// SIMATIC S7-200 project (STEP 7-Micro/WIN), CPU 224 UN REL 02.01

ORGANIZATION_BLOCK 主程序:OB1
TITLE=程序注释
BEGIN
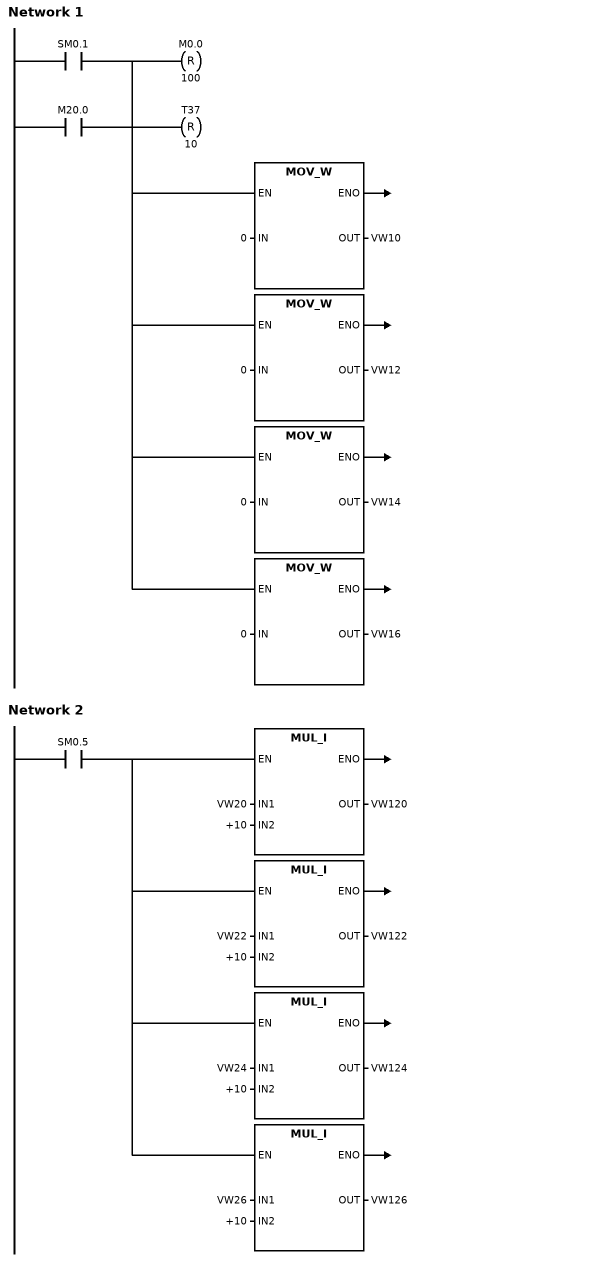
Network 1
LD     SM0.1
O      M20.0
R      M0.0, 100
R      T37, 10
MOVW   0, VW10
MOVW   0, VW12
MOVW   0, VW14
MOVW   0, VW16
Network 2
LD     SM0.5
MOVW   VW20, VW120
*I     +10, VW120
MOVW   VW22, VW122
*I     +10, VW122
MOVW   VW24, VW124
*I     +10, VW124
MOVW   VW26, VW126
*I     +10, VW126
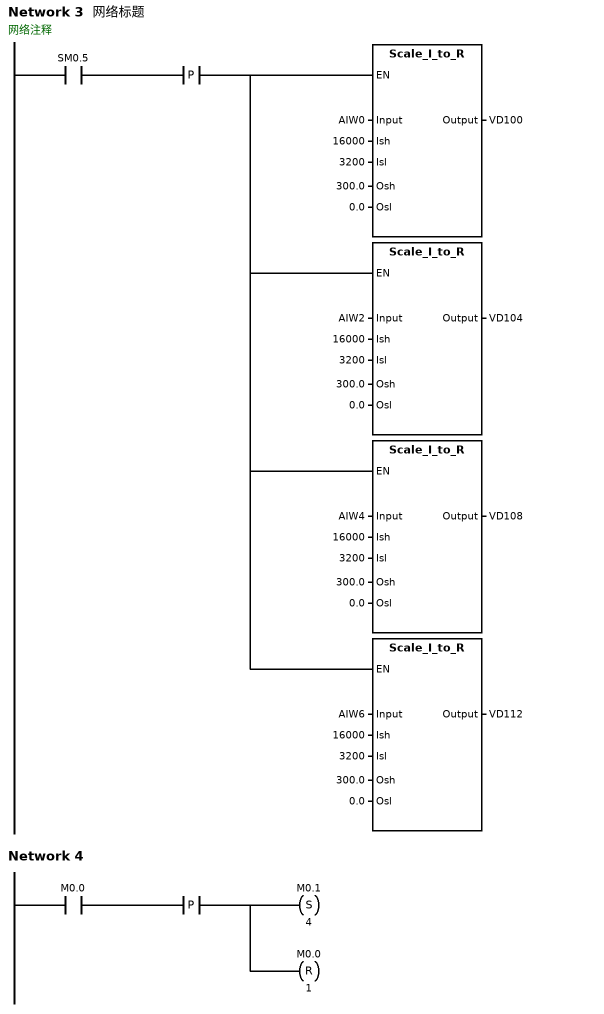
Network 3 // 网络标题
// 网络注释
LD     SM0.5
EU
CALL   Scale_I_to_R:SBR1, AIW0, 16000, 3200, 300.0, 0.0, VD100
CALL   Scale_I_to_R:SBR1, AIW2, 16000, 3200, 300.0, 0.0, VD104
CALL   Scale_I_to_R:SBR1, AIW4, 16000, 3200, 300.0, 0.0, VD108
CALL   Scale_I_to_R:SBR1, AIW6, 16000, 3200, 300.0, 0.0, VD112
Network 4
LD     M0.0
EU
S      M0.1, 4
R      M0.0, 1
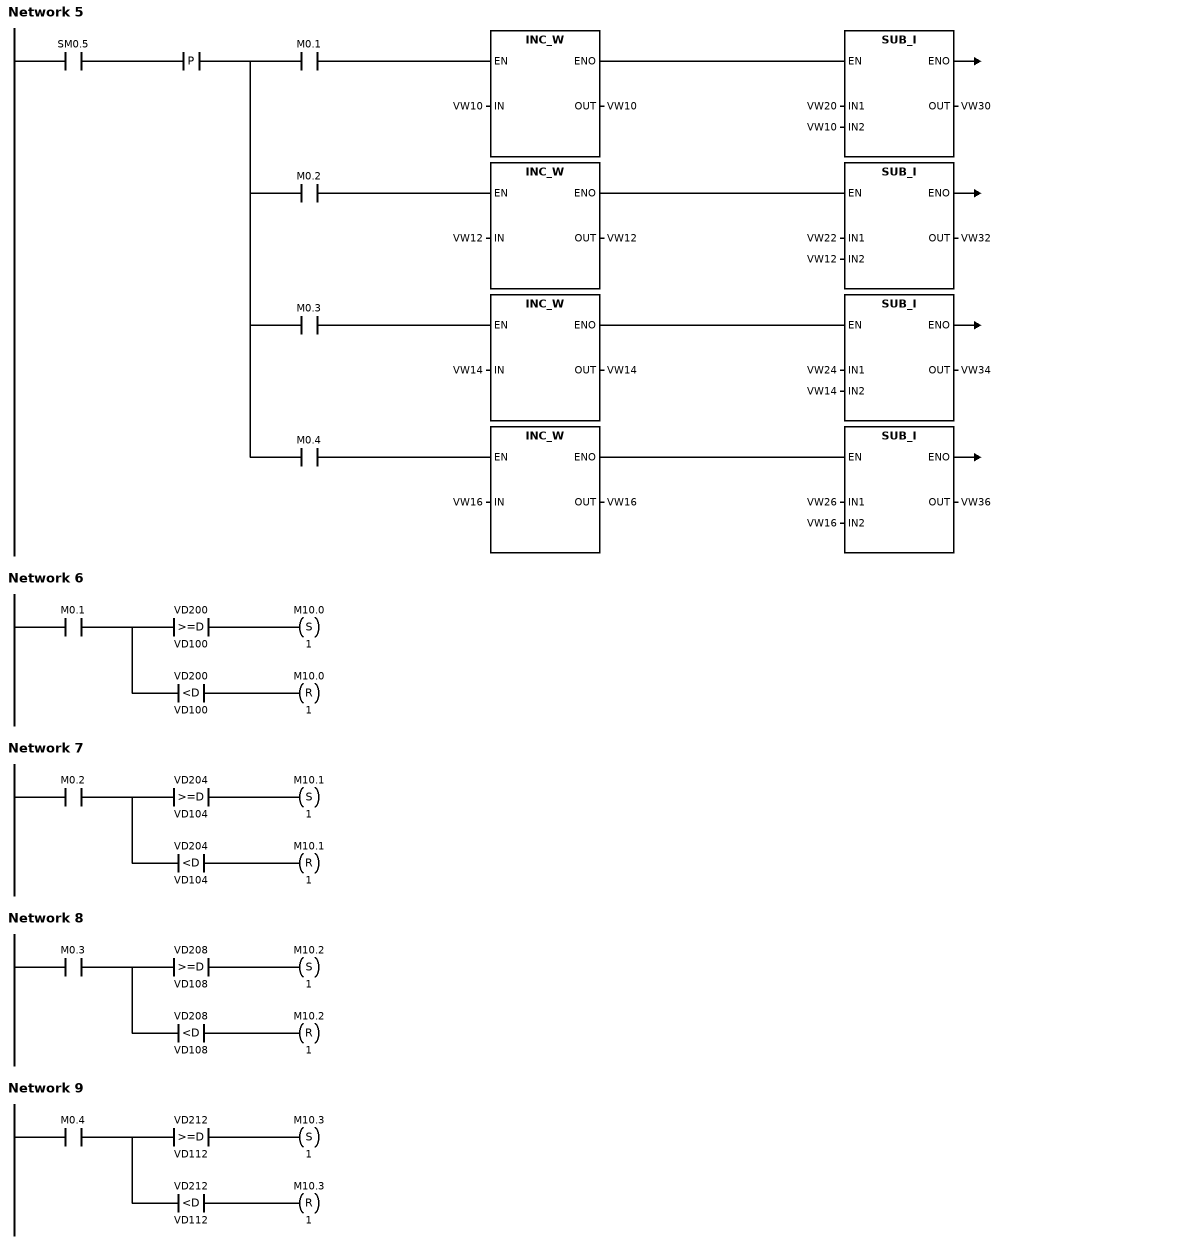
Network 5
LD     SM0.5
EU
LPS
A      M0.1
INCW   VW10
AENO
MOVW   VW20, VW30
-I     VW10, VW30
LRD
A      M0.2
INCW   VW12
AENO
MOVW   VW22, VW32
-I     VW12, VW32
LRD
A      M0.3
INCW   VW14
AENO
MOVW   VW24, VW34
-I     VW14, VW34
LPP
A      M0.4
INCW   VW16
AENO
MOVW   VW26, VW36
-I     VW16, VW36
Network 6
LD     M0.1
LPS
AD>=   VD200, VD100
S      M10.0, 1
LPP
AD<    VD200, VD100
R      M10.0, 1
Network 7
LD     M0.2
LPS
AD>=   VD204, VD104
S      M10.1, 1
LPP
AD<    VD204, VD104
R      M10.1, 1
Network 8
LD     M0.3
LPS
AD>=   VD208, VD108
S      M10.2, 1
LPP
AD<    VD208, VD108
R      M10.2, 1
Network 9
LD     M0.4
LPS
AD>=   VD212, VD112
S      M10.3, 1
LPP
AD<    VD212, VD112
R      M10.3, 1
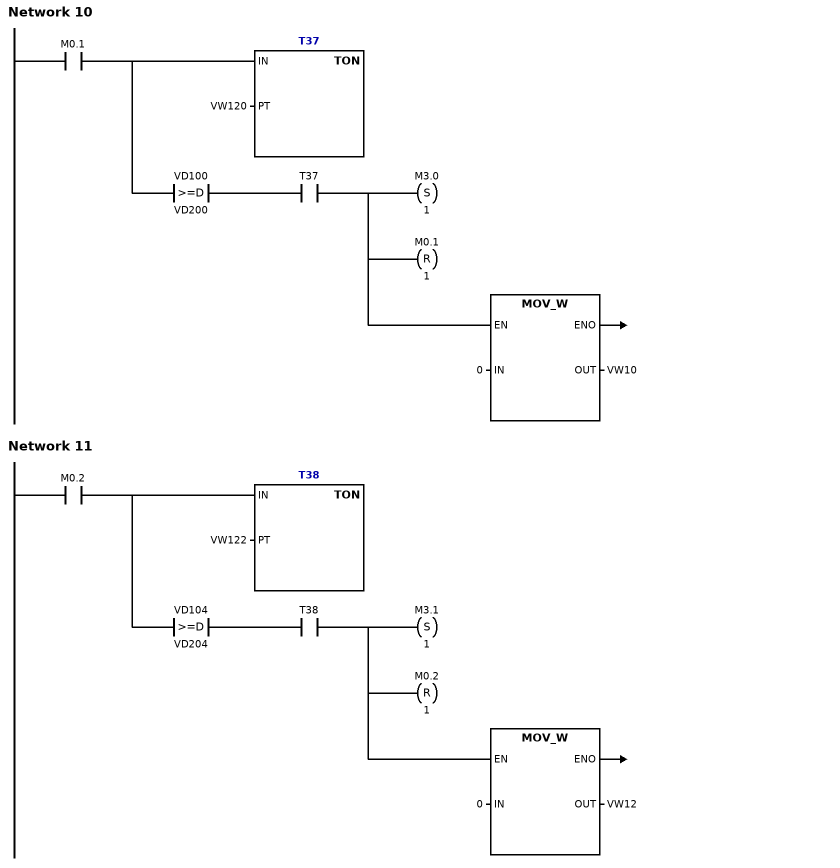
Network 10
LD     M0.1
TON    T37, VW120
AD>=   VD100, VD200
A      T37
S      M3.0, 1
R      M0.1, 1
MOVW   0, VW10
Network 11
LD     M0.2
TON    T38, VW122
AD>=   VD104, VD204
A      T38
S      M3.1, 1
R      M0.2, 1
MOVW   0, VW12
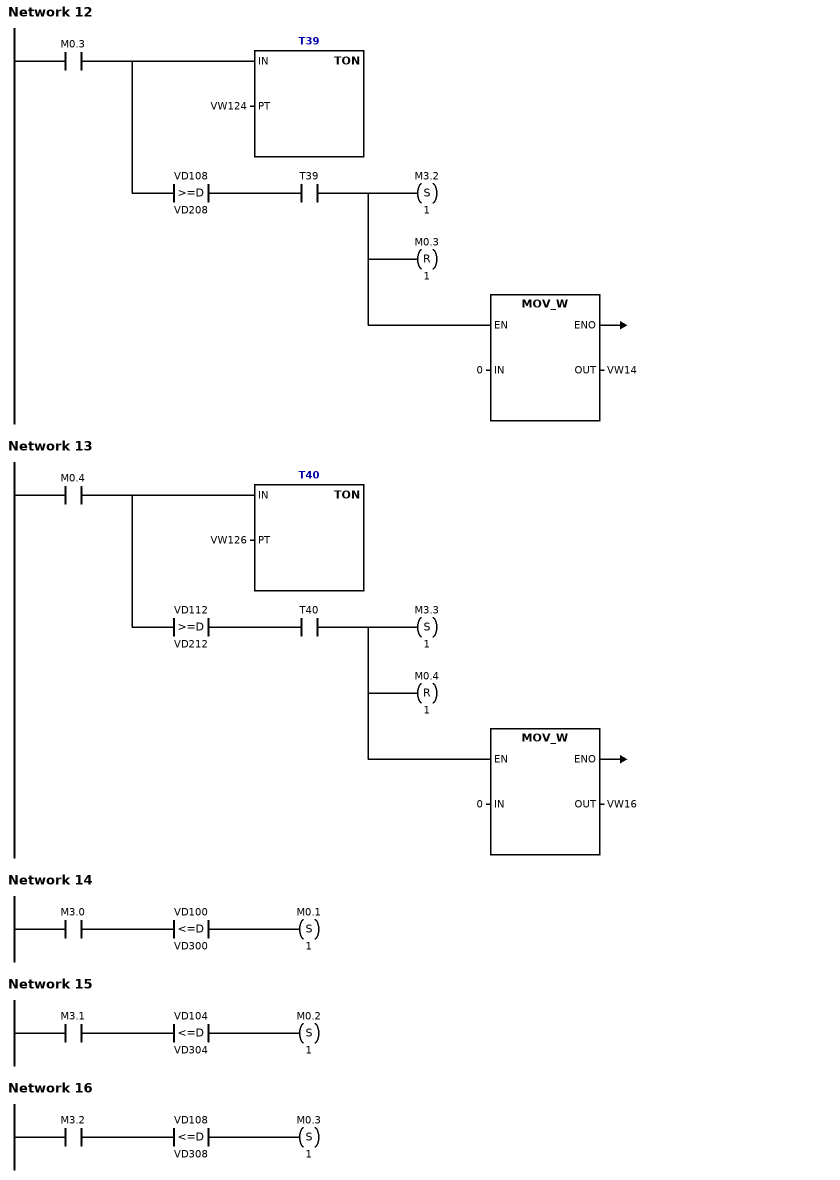
Network 12
LD     M0.3
TON    T39, VW124
AD>=   VD108, VD208
A      T39
S      M3.2, 1
R      M0.3, 1
MOVW   0, VW14
Network 13
LD     M0.4
TON    T40, VW126
AD>=   VD112, VD212
A      T40
S      M3.3, 1
R      M0.4, 1
MOVW   0, VW16
Network 14
LD     M3.0
AD<=   VD100, VD300
S      M0.1, 1
Network 15
LD     M3.1
AD<=   VD104, VD304
S      M0.2, 1
Network 16
LD     M3.2
AD<=   VD108, VD308
S      M0.3, 1
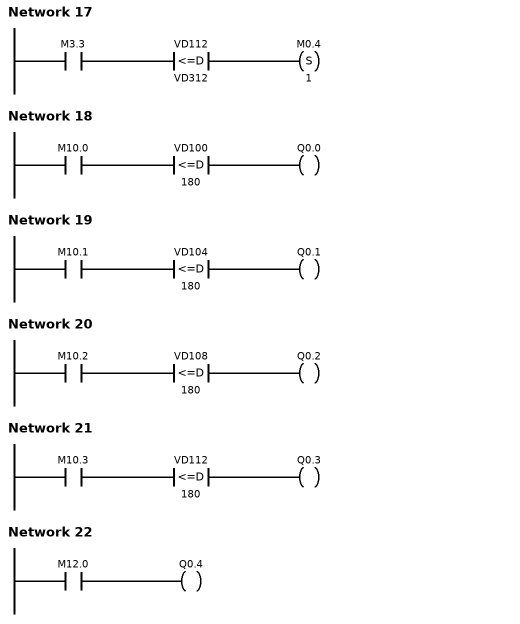
Network 17
LD     M3.3
AD<=   VD112, VD312
S      M0.4, 1
Network 18
LD     M10.0
AD<=   VD100, 180
=      Q0.0
Network 19
LD     M10.1
AD<=   VD104, 180
=      Q0.1
Network 20
LD     M10.2
AD<=   VD108, 180
=      Q0.2
Network 21
LD     M10.3
AD<=   VD112, 180
=      Q0.3
Network 22
LD     M12.0
=      Q0.4
END_ORGANIZATION_BLOCK

// SBR1: protected block, not included
